(*======================================================================================================================================*)
(*//=============================================================================\\
||  _   _ _  __  _         _                        _   _                      ||
|| | \ | | |/ / / \  _   _| |_ ___  _ __ ___   __ _| |_(_) ___  _ __         ||
|| |  \| | ' / / _ \| | | | __/ _ \| '_ ` _ \ / _` | __| |/ _ \| '_ \        ||
|| | |\  | . \/ ___ \ |_| | || (_) | | | | | | (_| | |_| | (_) | | | |       ||
|| |_| \_|_|\_\_/  \_\__,_|\__\___/|_| |_| |_|\__,_|\__|_|\___/|_| |_|       ||
||                                                                             ||
\\=============================================================================//
fb_RS485HB_StringBuilder:	Funktionsbaustein zum zusammenbauen komplexer Strings für Hausbus RS485 Ascii Telegramme		*)
(*
Date          	| Version    	| created under        	| Author          	| Remark *)
(*====================================================================================================================================================*)
(*22/01/2026   	| 1.00      	| TC3		  			| N.Kersting        | first release *)
(*22/01/2026   	| 1.01      	| TC3		  			| N.Kersting        | Erweiterung Array auf 8 Index *)
(*====================================================================================================================================================*)
FUNCTION_BLOCK fb_RS485HB_StringBuilder
VAR_INPUT
	I_bExecute			:BOOL := FALSE;
	I_diID				:DINT;				(* Device ID ( Steht auf dem Aufkleber und wird zur Identifizierung im BUS benötigt)*)
	I_iInstID			:INT;				(* Instanz ID *)
	I_EnumHBUnitTX		:E_EnumHBUnitTX;	(* Unit *)
	I_EnumHBCmdTX		:E_EnumHBCmdTX;		(* Command *)
	I_iCnt				:INT;				(* Anzahl der zusammengefügten Befehle *)
	I_iP1				:ARRAY[1..8] OF INT;				(* Parameter 1 *)
	I_iP2				:ARRAY[1..8] OF INT;				(* Parameter 2 *)
	I_iP3				:ARRAY[1..8] OF INT;				(* Parameter 3 *)
	I_iP4				:ARRAY[1..8] OF INT;				(* Parameter 4 *)
END_VAR
VAR_OUTPUT	
	Q_sOut				:STRING(255);							(* Fertiger Ausgabestring*)	
	Q_bDone				:BOOL;
	Q_bError			:BOOL;
END_VAR
VAR
	IDX 				:INT;
	Trig				:r_trig;
	nLength				:INT;
END_VAR

Trig(CLK:=I_bExecute);

IF Trig.Q
	AND I_bExecute
THEN
	IF I_diID <> 0
	THEN
		IF I_iInstID <> 0
		THEN
			IF I_iCnt <>0
				AND I_iCnt <=8
			THEN
				Q_bError := FALSE;
				
				CASE I_iCnt OF
				(*===========================*)
				0: 	IDX := 0;
					Q_sOut :='';
					
					Q_bDone := TRUE;
					RETURN;
					
				(*===========================*)
				1: 	IDX := 1;
					Q_sOut 	:=		F_RS485HB_TO_ASCII(I_diID,I_iInstID,I_EnumHBUnitTX,I_EnumHBCmdTX,I_iP1[IDX],I_iP2[IDX],I_iP3[IDX],I_iP4[IDX]);
					
					Q_bDone := TRUE;
					
				(*===========================*)
				2: 	IDX := 1;
					Q_sOut 	:=		F_RS485HB_TO_ASCII(I_diID,I_iInstID,I_EnumHBUnitTX,I_EnumHBCmdTX,I_iP1[IDX],I_iP2[IDX],I_iP3[IDX],I_iP4[IDX]);
					IDX := 2;
					Q_sOut 	:=		CONCAT(Q_sOut,F_RS485HB_TO_ASCII(I_diID,I_iInstID+IDX-1,I_EnumHBUnitTX,I_EnumHBCmdTX,I_iP1[IDX],I_iP2[IDX],I_iP3[IDX],I_iP4[IDX]));
					
					Q_bDone := TRUE;
					
				(*===========================*)
				3: 	IDX := 1;
					Q_sOut 	:=		F_RS485HB_TO_ASCII(I_diID,I_iInstID,I_EnumHBUnitTX,I_EnumHBCmdTX,I_iP1[IDX],I_iP2[IDX],I_iP3[IDX],I_iP4[IDX]);
					IDX := 2;
					Q_sOut 	:=		CONCAT(Q_sOut,F_RS485HB_TO_ASCII(I_diID,I_iInstID+IDX-1,I_EnumHBUnitTX,I_EnumHBCmdTX,I_iP1[IDX],I_iP2[IDX],I_iP3[IDX],I_iP4[IDX]));
					IDX := 3;
					Q_sOut 	:=		CONCAT(Q_sOut,F_RS485HB_TO_ASCII(I_diID,I_iInstID+IDX-1,I_EnumHBUnitTX,I_EnumHBCmdTX,I_iP1[IDX],I_iP2[IDX],I_iP3[IDX],I_iP4[IDX]));
					
					Q_bDone := TRUE;
					
				(*===========================*)
				4: 	IDX := 1;
					Q_sOut 	:=		F_RS485HB_TO_ASCII(I_diID,I_iInstID,I_EnumHBUnitTX,I_EnumHBCmdTX,I_iP1[IDX],I_iP2[IDX],I_iP3[IDX],I_iP4[IDX]);
					IDX := 2;
					Q_sOut 	:=		CONCAT(Q_sOut,F_RS485HB_TO_ASCII(I_diID,I_iInstID+IDX-1,I_EnumHBUnitTX,I_EnumHBCmdTX,I_iP1[IDX],I_iP2[IDX],I_iP3[IDX],I_iP4[IDX]));
					IDX := 3;
					Q_sOut 	:=		CONCAT(Q_sOut,F_RS485HB_TO_ASCII(I_diID,I_iInstID+IDX-1,I_EnumHBUnitTX,I_EnumHBCmdTX,I_iP1[IDX],I_iP2[IDX],I_iP3[IDX],I_iP4[IDX]));
					IDX := 4;
					Q_sOut 	:=		CONCAT(Q_sOut,F_RS485HB_TO_ASCII(I_diID,I_iInstID+IDX-1,I_EnumHBUnitTX,I_EnumHBCmdTX,I_iP1[IDX],I_iP2[IDX],I_iP3[IDX],I_iP4[IDX]));
					
					Q_bDone := TRUE;
					
				(*===========================*)
				5: 	IDX := 1;
					Q_sOut 	:=		F_RS485HB_TO_ASCII(I_diID,I_iInstID,I_EnumHBUnitTX,I_EnumHBCmdTX,I_iP1[IDX],I_iP2[IDX],I_iP3[IDX],I_iP4[IDX]);
					IDX := 2;
					Q_sOut 	:=		CONCAT(Q_sOut,F_RS485HB_TO_ASCII(I_diID,I_iInstID+IDX-1,I_EnumHBUnitTX,I_EnumHBCmdTX,I_iP1[IDX],I_iP2[IDX],I_iP3[IDX],I_iP4[IDX]));
					IDX := 3;
					Q_sOut 	:=		CONCAT(Q_sOut,F_RS485HB_TO_ASCII(I_diID,I_iInstID+IDX-1,I_EnumHBUnitTX,I_EnumHBCmdTX,I_iP1[IDX],I_iP2[IDX],I_iP3[IDX],I_iP4[IDX]));
					IDX := 4;
					Q_sOut 	:=		CONCAT(Q_sOut,F_RS485HB_TO_ASCII(I_diID,I_iInstID+IDX-1,I_EnumHBUnitTX,I_EnumHBCmdTX,I_iP1[IDX],I_iP2[IDX],I_iP3[IDX],I_iP4[IDX]));
					IDX := 5;
					Q_sOut 	:=		CONCAT(Q_sOut,F_RS485HB_TO_ASCII(I_diID,I_iInstID+IDX-1,I_EnumHBUnitTX,I_EnumHBCmdTX,I_iP1[IDX],I_iP2[IDX],I_iP3[IDX],I_iP4[IDX]));
					
					Q_bDone := TRUE;
					
				(*===========================*)
				6: 	IDX := 1;
					Q_sOut 	:=		F_RS485HB_TO_ASCII(I_diID,I_iInstID,I_EnumHBUnitTX,I_EnumHBCmdTX,I_iP1[IDX],I_iP2[IDX],I_iP3[IDX],I_iP4[IDX]);
					IDX := 2;
					Q_sOut 	:=		CONCAT(Q_sOut,F_RS485HB_TO_ASCII(I_diID,I_iInstID+IDX-1,I_EnumHBUnitTX,I_EnumHBCmdTX,I_iP1[IDX],I_iP2[IDX],I_iP3[IDX],I_iP4[IDX]));
					IDX := 3;
					Q_sOut 	:=		CONCAT(Q_sOut,F_RS485HB_TO_ASCII(I_diID,I_iInstID+IDX-1,I_EnumHBUnitTX,I_EnumHBCmdTX,I_iP1[IDX],I_iP2[IDX],I_iP3[IDX],I_iP4[IDX]));
					IDX := 4;
					Q_sOut 	:=		CONCAT(Q_sOut,F_RS485HB_TO_ASCII(I_diID,I_iInstID+IDX-1,I_EnumHBUnitTX,I_EnumHBCmdTX,I_iP1[IDX],I_iP2[IDX],I_iP3[IDX],I_iP4[IDX]));
					IDX := 5;
					Q_sOut 	:=		CONCAT(Q_sOut,F_RS485HB_TO_ASCII(I_diID,I_iInstID+IDX-1,I_EnumHBUnitTX,I_EnumHBCmdTX,I_iP1[IDX],I_iP2[IDX],I_iP3[IDX],I_iP4[IDX]));
					IDX := 6;
					Q_sOut 	:=		CONCAT(Q_sOut,F_RS485HB_TO_ASCII(I_diID,I_iInstID+IDX-1,I_EnumHBUnitTX,I_EnumHBCmdTX,I_iP1[IDX],I_iP2[IDX],I_iP3[IDX],I_iP4[IDX]));
					
					Q_bDone := TRUE;
					
				(*===========================*)
				7: 	IDX := 1;
					Q_sOut 	:=		F_RS485HB_TO_ASCII(I_diID,I_iInstID,I_EnumHBUnitTX,I_EnumHBCmdTX,I_iP1[IDX],I_iP2[IDX],I_iP3[IDX],I_iP4[IDX]);
					IDX := 2;
					Q_sOut 	:=		CONCAT(Q_sOut,F_RS485HB_TO_ASCII(I_diID,I_iInstID+IDX-1,I_EnumHBUnitTX,I_EnumHBCmdTX,I_iP1[IDX],I_iP2[IDX],I_iP3[IDX],I_iP4[IDX]));
					IDX := 3;
					Q_sOut 	:=		CONCAT(Q_sOut,F_RS485HB_TO_ASCII(I_diID,I_iInstID+IDX-1,I_EnumHBUnitTX,I_EnumHBCmdTX,I_iP1[IDX],I_iP2[IDX],I_iP3[IDX],I_iP4[IDX]));
					IDX := 4;
					Q_sOut 	:=		CONCAT(Q_sOut,F_RS485HB_TO_ASCII(I_diID,I_iInstID+IDX-1,I_EnumHBUnitTX,I_EnumHBCmdTX,I_iP1[IDX],I_iP2[IDX],I_iP3[IDX],I_iP4[IDX]));
					IDX := 5;
					Q_sOut 	:=		CONCAT(Q_sOut,F_RS485HB_TO_ASCII(I_diID,I_iInstID+IDX-1,I_EnumHBUnitTX,I_EnumHBCmdTX,I_iP1[IDX],I_iP2[IDX],I_iP3[IDX],I_iP4[IDX]));
					IDX := 6;
					Q_sOut 	:=		CONCAT(Q_sOut,F_RS485HB_TO_ASCII(I_diID,I_iInstID+IDX-1,I_EnumHBUnitTX,I_EnumHBCmdTX,I_iP1[IDX],I_iP2[IDX],I_iP3[IDX],I_iP4[IDX]));
					IDX := 7;
					Q_sOut 	:=		CONCAT(Q_sOut,F_RS485HB_TO_ASCII(I_diID,I_iInstID+IDX-1,I_EnumHBUnitTX,I_EnumHBCmdTX,I_iP1[IDX],I_iP2[IDX],I_iP3[IDX],I_iP4[IDX]));
					
					Q_bDone := TRUE;
				
				(*===========================*)
				8: 	IDX := 1;
					Q_sOut 	:=		F_RS485HB_TO_ASCII(I_diID,I_iInstID,I_EnumHBUnitTX,I_EnumHBCmdTX,I_iP1[IDX],I_iP2[IDX],I_iP3[IDX],I_iP4[IDX]);
					IDX := 2;
					Q_sOut 	:=		CONCAT(Q_sOut,F_RS485HB_TO_ASCII(I_diID,I_iInstID+IDX-1,I_EnumHBUnitTX,I_EnumHBCmdTX,I_iP1[IDX],I_iP2[IDX],I_iP3[IDX],I_iP4[IDX]));
					IDX := 3;
					Q_sOut 	:=		CONCAT(Q_sOut,F_RS485HB_TO_ASCII(I_diID,I_iInstID+IDX-1,I_EnumHBUnitTX,I_EnumHBCmdTX,I_iP1[IDX],I_iP2[IDX],I_iP3[IDX],I_iP4[IDX]));
					IDX := 4;
					Q_sOut 	:=		CONCAT(Q_sOut,F_RS485HB_TO_ASCII(I_diID,I_iInstID+IDX-1,I_EnumHBUnitTX,I_EnumHBCmdTX,I_iP1[IDX],I_iP2[IDX],I_iP3[IDX],I_iP4[IDX]));
					IDX := 5;
					Q_sOut 	:=		CONCAT(Q_sOut,F_RS485HB_TO_ASCII(I_diID,I_iInstID+IDX-1,I_EnumHBUnitTX,I_EnumHBCmdTX,I_iP1[IDX],I_iP2[IDX],I_iP3[IDX],I_iP4[IDX]));
					IDX := 6;
					Q_sOut 	:=		CONCAT(Q_sOut,F_RS485HB_TO_ASCII(I_diID,I_iInstID+IDX-1,I_EnumHBUnitTX,I_EnumHBCmdTX,I_iP1[IDX],I_iP2[IDX],I_iP3[IDX],I_iP4[IDX]));
					IDX := 7;
					Q_sOut 	:=		CONCAT(Q_sOut,F_RS485HB_TO_ASCII(I_diID,I_iInstID+IDX-1,I_EnumHBUnitTX,I_EnumHBCmdTX,I_iP1[IDX],I_iP2[IDX],I_iP3[IDX],I_iP4[IDX]));
					IDX := 8;
					Q_sOut 	:=		CONCAT(Q_sOut,F_RS485HB_TO_ASCII(I_diID,I_iInstID+IDX-1,I_EnumHBUnitTX,I_EnumHBCmdTX,I_iP1[IDX],I_iP2[IDX],I_iP3[IDX],I_iP4[IDX]));
					
					Q_bDone := TRUE;	
				END_CASE
				
				nLength :=	LEN(Q_sOut);
				RETURN;
			ELSE
				Q_bError := TRUE;
			END_IF
		ELSE
			Q_bError := TRUE;
		END_IF
	ELSE
		Q_bError := TRUE;
	END_IF
ELSIF
	NOT I_bExecute
THEN
	Q_bDone := FALSE;
	Q_sOut :='x';
END_IF

END_FUNCTION_BLOCK

(* stored: Version 1.1.0.1, ProductVersion 3.1.4024.15
   POU fb_RS485HB_StringBuilder: Id {f075a23d-6b83-49cb-bbeb-d93ad99a9ff1}, SpecialFunc None *)
